PROGRAM MAIN
VAR
	initialized : BOOL := FALSE;
	
	stThisIsFirstInstanceOfAStructure : ST_Event;

	eEventType : E_EventType := E_EventType.Alarm;
	eEventSeverity : TcEventSeverity := TcEventSeverity.Info;
	nEventIdentity : UDINT := 44444;
	sEventText : STRING(255) := 'Some informational event';
	
//	CsvPersistentEventStorage : FB_CsvPersistentEventStorage;
//	EventLogger : EventLogger(CsvPersistentEventStorage);

		arr1 : ARRAY[1..3] OF BOOL;
		arr2 : ARRAY[1..3] OF BOOL;
		arr3 : ARRAY[1..3] OF BOOL;
		arr4 : ARRAY[1..3] OF BOOL;
		
		
		arr5 : ARRAY[1..2] OF BOOL;
		arr6 : ARRAY[1..2] OF BOOL;
		
		//button1 : LightSwitch;//ShutterSwitch;//LightSwitch;//UpStopDownButton;// LightSwitch;	
		button2 : ShutterSwitch;
	isDay : BOOL := TRUE;
	minimumLogSeverity : TcEventSeverity := TcEventSeverity.Verbose;
END_VAR

VAR_IN_OUT

END_VAR

IF NOT initialized THEN
	GVL.EventLogger.print1(level:=TcEventSeverity.Info, str1:='PLC started');
	initButtons();	

			F_UpdateEventTimestampWithSystemTime(stEvent := stThisIsFirstInstanceOfAStructure);	
			GVL.EventLogger.AddEvent(eEventType, eEventSeverity, nEventIdentity, sEventText);
			
	initialized := TRUE;
END_IF


//-------------------------------

//CsvPersistentEventStorage();


button2.loop();

METHOD initButtons
VAR_INPUT
END_VAR
button2(ID:= 1,	digitalInputUp:= GVL.b_button_4,	digitalInputDown:= GVL.b_button_5,down_outputs:=arr5, up_outputs:=arr6); //shutter switch
 
//button1(ID := 1, digitalInput := GVL.b_button_4, small_outputs := arr1,	medium_outputs := arr2,	big_outputs := arr3,
//	superstrong_outputs := arr4, 	levelsManaged := 4,	defaultDayOutput := E_OutputLevel.big,	defaultNightOutput := E_OutputLevel.small); //light switch
	
	
//button1(ID:= 1, digitalInput := GVL.b_button_4, outputs := arr1, defaultFirstClickDirection := E_Direction.UP);
	
//button1(digitalInput:= GVL.b_button_4, ID:=1, name:='goscinny', outputs := arr1, runAsYouPress := FALSE);
END_METHOD

END_PROGRAM

(* stored: Version 1.1.0.1, ProductVersion 3.1.4024.12
   POU MAIN: Id {ba37e07b-b35e-420a-a01b-24b84cc886a6}, SpecialFunc None
   Method initButtons: Id {bf7480a3-2217-4091-9e5a-54e832bdb26c} *)
